FUNCTION_BLOCK MOD_StateView (* The module's PackML state from its local channel; asks for the current value at INIT *)
  (* Standard: 61499-2 *)
  (* Version 0.1, 2026-09-28, Project contributors, AAU Smart Production Lab *)
  PACKAGE modlib;
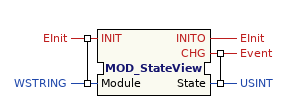
  EVENT_INPUT
    INIT : EInit WITH Module;
  END_EVENT
  EVENT_OUTPUT
    INITO : EInit;
    CHG WITH State;
  END_EVENT
  VAR_INPUT
    Module : WSTRING;
  END_VAR
  VAR_OUTPUT
    State : USINT;
  END_VAR
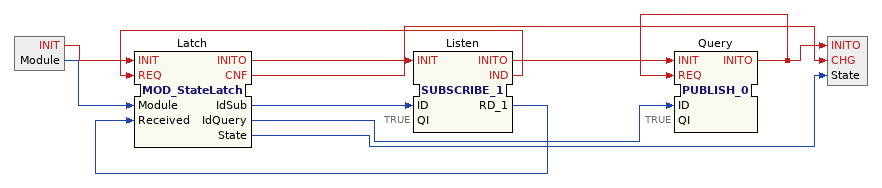
  FBS
    Latch : modlib::MOD_StateLatch;
    Listen : iec61499::net::SUBSCRIBE_1(QI := TRUE);
    Query : iec61499::net::PUBLISH_0(QI := TRUE);
  END_FBS
  EVENT_CONNECTIONS
    INIT TO Latch.INIT;
    Latch.INITO TO Listen.INIT;
    Listen.INITO TO Query.INIT;
    Query.INITO TO Query.REQ;
    Query.INITO TO INITO;
    Listen.IND TO Latch.REQ;
    Latch.CNF TO CHG;
  END_CONNECTIONS
  DATA_CONNECTIONS
    Module TO Latch.Module;
    Latch.IdSub TO Listen.ID;
    Latch.IdQuery TO Query.ID;
    Listen.RD_1 TO Latch.Received;
    Latch.State TO State;
  END_CONNECTIONS
END_FUNCTION_BLOCK
